FUNCTION_BLOCK FB_Station
VAR
	stUnitArr			: ARRAY [1..100] OF ST_Unit;
	iMaxUnit			: INT;
	iLastIndex			: INT;
	
	iMaxLevel			: INT;
	iCurLevel			: INT := 1;
	
	rLocation			: REAL;
END_VAR

PROPERTY HasChicken : BOOL
GET
VAR
	iIndex			: INT;
END_VAR
HasChicken := FALSE;
IF iLastIndex > 0 THEN
	FOR iIndex := 1 TO iLastIndex BY 1 DO
		IF stUnitArr[iIndex].eType = 1 THEN
			HasChicken := NOT HasChicken;
			RETURN;
		END_IF
	END_FOR
END_IF
END_GET
END_PROPERTY

PROPERTY HasEgg : BOOL
GET
VAR
	iIndex			: INT;
END_VAR
HasEgg := FALSE;
IF iLastIndex > 0 THEN
	FOR iIndex := 1 TO iLastIndex BY 1 DO
		IF stUnitArr[iIndex].eType = 0 THEN
			HasEgg := NOT HasEgg;
			RETURN;
		END_IF
	END_FOR
END_IF
END_GET
END_PROPERTY

METHOD HpDeduct : PVOID
VAR
	iTempIndex			: INT;
END_VAR
IF iLastIndex < 1 THEN
	RETURN;
END_IF

FOR iTempIndex := 1 TO iLastIndex BY 1 DO
	stUnitArr[iTempIndex].iHitPoint := stUnitArr[iTempIndex].iHitPoint - 1;
	IF stUnitArr[iTempIndex].iHitPoint = 0 THEN
		RemoveUnit(iTempIndex);
	END_IF
END_FOR
END_METHOD

METHOD HpRecover : PVOID
VAR
	iTempIndex			: INT;
END_VAR
IF iLastIndex < 1 THEN
	RETURN;
END_IF

FOR iTempIndex := 1 TO iLastIndex BY 1 DO
	IF stUnitArr[iTempIndex].iHitPoint < 30 THEN
		stUnitArr[iTempIndex].iHitPoint := stUnitArr[iTempIndex].iHitPoint + 1;
	END_IF
END_FOR
END_METHOD

PROPERTY IsFull : BOOL
GET
IsFull := TRUE;
IF iLastIndex < iMaxUnit THEN
	IsFull := NOT IsFull;
END_IF
END_GET
END_PROPERTY

PROPERTY Level : INT
GET
Level := iCurLevel;
END_GET
END_PROPERTY

PROPERTY Location : REAL
GET
Location := rLocation;
END_GET
END_PROPERTY

METHOD RemoveUnit : PVOID
VAR_INPUT
	iIndex			: INT;
END_VAR
stUnitArr[iIndex] := stUnitArr[iLastIndex];
stUnitArr[iLastIndex].eType := -1;
stUnitArr[iLastIndex].iHitPoint := 0;
stUnitArr[iLastIndex].iProgress := 0;
iLastIndex := iLastIndex - 1;
END_METHOD

METHOD Run : BOOL
VAR_INPUT
END_VAR
iMaxUnit := iCurLevel * 10;
END_METHOD

METHOD Set : PVOID
VAR_INPUT
	MaxLevel			: INT;
	Location			: REAL;
END_VAR
iMaxLevel := MaxLevel;
rLocation := Location;
iCurLevel := 1;
END_METHOD

METHOD SortAscending : PVOID
VAR
	iCurIndex			: INT;
	stTempUnit			: ST_Unit;
	iTempIndex			: INT;
END_VAR
IF iLastIndex < 2 THEN
	RETURN;
END_IF

FOR iTempIndex := 1 TO iLastIndex BY 1 DO
	FOR iCurIndex := 1 TO iLastIndex BY 1 DO
		IF stUnitArr[iCurIndex].iHitPoint > stUnitArr[iTempIndex].iHitPoint THEN
			stTempUnit := stUnitArr[iCurIndex];
			stUnitArr[iCurIndex] := stUnitArr[iTempIndex];
			stUnitArr[iTempIndex] := stTempUnit;
		END_IF
	END_FOR
END_FOR
END_METHOD

METHOD SortDescending : PVOID
VAR
	iCurIndex			: INT;
	stTempUnit			: ST_Unit;
	iTempIndex			: INT;
END_VAR
IF iLastIndex < 2 THEN
	RETURN;
END_IF

FOR iTempIndex := 1 TO iLastIndex BY 1 DO
	FOR iCurIndex := 1 TO iLastIndex BY 1 DO
		IF stUnitArr[iCurIndex].iHitPoint < stUnitArr[iTempIndex].iHitPoint THEN
			stTempUnit := stUnitArr[iCurIndex];
			stUnitArr[iCurIndex] := stUnitArr[iTempIndex];
			stUnitArr[iTempIndex] := stTempUnit;
		END_IF
	END_FOR
END_FOR
END_METHOD

PROPERTY TotalUnit : INT
GET
TotalUnit := iLastIndex;
END_GET
END_PROPERTY

METHOD UnitExport : ST_Unit
VAR_INPUT
	UnitType			: INT; // 0: Egg, 1: Chicken
END_VAR
VAR
	iTempIndex			: INT;
END_VAR
IF iLastIndex < 1 THEN
	RETURN;
END_IF

CASE UnitType OF
	0: 
		FOR iTempIndex := 1 TO iLastIndex BY 1 DO
			IF stUnitArr[iTempIndex].eType = UnitType THEN
				stUnitArr[iTempIndex].iProgress := 0;
				UnitExport := stUnitArr[iTempIndex];
				stUnitArr[iTempIndex] := stUnitArr[iLastIndex];
				stUnitArr[iLastIndex].eType := -1;
				stUnitArr[iLastIndex].iHitPoint := 0;
				iLastIndex := iLastIndex - 1;
				RETURN;
			END_IF
		END_FOR
		
	1:
		FOR iTempIndex := 1 TO iLastIndex BY 1 DO
			IF stUnitArr[iTempIndex].eType = UnitType THEN
				stUnitArr[iTempIndex].iProgress := 0;
				UnitExport := stUnitArr[iTempIndex];
				stUnitArr[iTempIndex] := stUnitArr[iLastIndex];
				stUnitArr[iLastIndex].eType := -1;
				stUnitArr[iLastIndex].iHitPoint := 0;
				iLastIndex := iLastIndex - 1;
				RETURN;
			END_IF
		END_FOR
END_CASE
END_METHOD

METHOD UnitImport : PVOID
VAR_INPUT
	Unit			: ST_Unit;
END_VAR
IF Unit.eType <> -1 THEN
	IF iLastIndex < iMaxUnit THEN
		iLastIndex := iLastIndex + 1;
		stUnitArr[iLastIndex] := Unit;
	END_IF
END_IF
END_METHOD

METHOD Upgrade : PVOID
IF iCurLevel < iMaxLevel THEN
	iCurLevel := iCurLevel + 1;
END_IF
END_METHOD

END_FUNCTION_BLOCK

(* stored: Version 1.1.0.1, ProductVersion 3.1.4024.12
   POU FB_Station: Id {fa9608f7-10b1-49a0-93c0-54a46514fd0d}, SpecialFunc None
   Folder Properties: Id {cbf9eb36-f301-4eff-929e-8c86fc0f2250}
   Property HasChicken: Id {c93ed1ef-3654-47cb-aa24-135c3c4f942d}
   Get Get: Id {4be2f8ba-4fa3-450c-b7ac-7bbba6d7084e}
   Property HasEgg: Id {b140493c-7e54-4932-a2b3-a290ab1e592b}
   Get Get: Id {64f83d36-90c4-4942-aa6c-681bd7c09926}
   Method HpDeduct: Id {85e37be9-392a-462c-bf3b-e2daa26ec517}
   Method HpRecover: Id {f06cad78-0f1e-4abe-978b-f240cdfab569}
   Property IsFull: Id {e7fe457d-fa78-4d80-91a3-3ca9cd53af44}
   Get Get: Id {ff251fa9-273a-4834-ba24-a217c2905242}
   Property Level: Id {1e558226-5e6a-4228-836a-c1984b49fda3}
   Get Get: Id {40b1a418-8c16-4d1f-b09c-d9dcb7205473}
   Property Location: Id {dfc70d4f-c752-4532-9b94-56931eabe2a5}
   Get Get: Id {251ac9ff-8af7-4cf7-81c5-5f8d0b1a6186}
   Method RemoveUnit: Id {0dc9de5b-c854-46f7-baa7-f6cad565c0e8}
   Method Run: Id {29adece8-1a8b-4c56-8ca4-ad76a7e2a383}
   Method Set: Id {859eb24e-bd03-4a04-b53f-b0941150ff0c}
   Method SortAscending: Id {81cc50fa-f286-4208-a120-5248de96850f}
   Method SortDescending: Id {4d2ef8e1-06aa-40b5-8dcb-502a6dcf2298}
   Property TotalUnit: Id {2c8335a1-57c5-4d23-9140-156d3c02720b}
   Get Get: Id {b7c489f8-94b4-4068-aeaa-0dc12d125db8}
   Method UnitExport: Id {ab8aafad-4c05-4c03-91cb-69140f668fcd}
   Method UnitImport: Id {b9b1ce72-efa1-4e57-bb72-c0809f7cfc8a}
   Method Upgrade: Id {58a8775b-8909-4efa-afa5-d70add47deb0} *)
